// Mitsubishi GX Works2 project: MasterPlc3_2   PLC: Q03UDE

PROGRAM OUTPUT
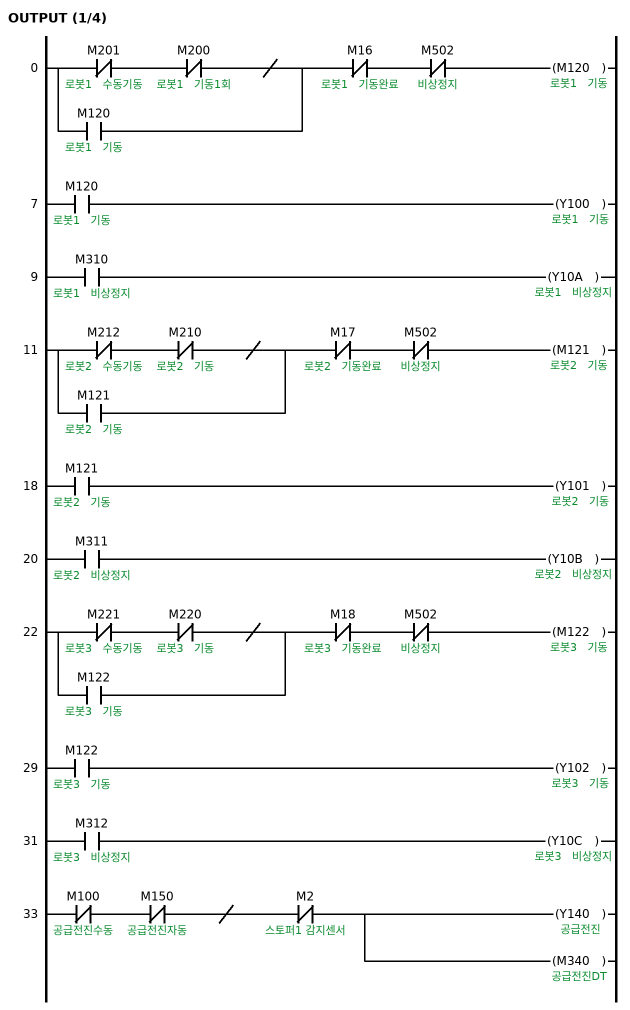
0     LDI     M201  ; 로봇1   수동기동
      ANI     M200  ; 로봇1   기동1회
      INV
      OR      M120  ; 로봇1   기동
      ANI     M16  ; 로봇1   기동완료
      ANI     M502  ; 비상정지
      OUT     M120  ; 로봇1   기동
7     LD      M120  ; 로봇1   기동
      OUT     Y100  ; 로봇1   기동
9     LD      M310  ; 로봇1   비상정지
      OUT     Y10A  ; 로봇1   비상정지
11    LDI     M212  ; 로봇2   수동기동
      ANI     M210  ; 로봇2   기동
      INV
      OR      M121  ; 로봇2   기동
      ANI     M17  ; 로봇2   기동완료
      ANI     M502  ; 비상정지
      OUT     M121  ; 로봇2   기동
18    LD      M121  ; 로봇2   기동
      OUT     Y101  ; 로봇2   기동
20    LD      M311  ; 로봇2   비상정지
      OUT     Y10B  ; 로봇2   비상정지
22    LDI     M221  ; 로봇3   수동기동
      ANI     M220  ; 로봇3   기동
      INV
      OR      M122  ; 로봇3   기동
      ANI     M18  ; 로봇3   기동완료
      ANI     M502  ; 비상정지
      OUT     M122  ; 로봇3   기동
29    LD      M122  ; 로봇3   기동
      OUT     Y102  ; 로봇3   기동
31    LD      M312  ; 로봇3   비상정지
      OUT     Y10C  ; 로봇3   비상정지
33    LDI     M100  ; 공급전진수동
      ANI     M150  ; 공급전진자동
      INV
      ANI     M2  ; 스토퍼1 감지센서
      OUT     Y140  ; 공급전진
      OUT     M340  ; 공급전진DT
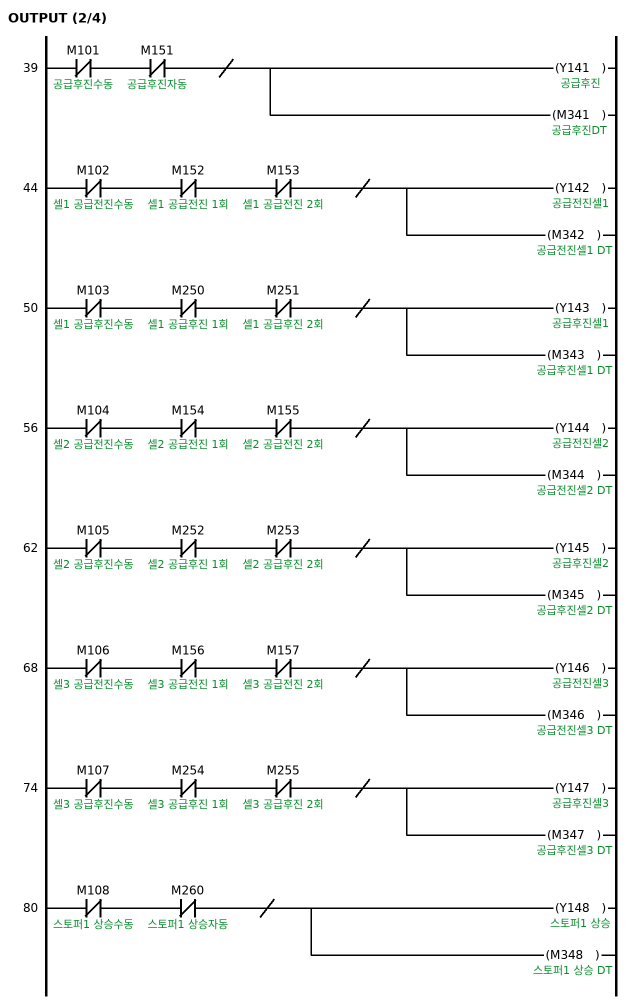
39    LDI     M101  ; 공급후진수동
      ANI     M151  ; 공급후진자동
      INV
      OUT     Y141  ; 공급후진
      OUT     M341  ; 공급후진DT
44    LDI     M102  ; 셀1 공급전진수동
      ANI     M152  ; 셀1 공급전진 1회
      ANI     M153  ; 셀1 공급전진 2회
      INV
      OUT     Y142  ; 공급전진셀1
      OUT     M342  ; 공급전진셀1 DT
50    LDI     M103  ; 셀1 공급후진수동
      ANI     M250  ; 셀1 공급후진 1회
      ANI     M251  ; 셀1 공급후진 2회
      INV
      OUT     Y143  ; 공급후진셀1
      OUT     M343  ; 공급후진셀1 DT
56    LDI     M104  ; 셀2 공급전진수동
      ANI     M154  ; 셀2 공급전진 1회
      ANI     M155  ; 셀2 공급전진 2회
      INV
      OUT     Y144  ; 공급전진셀2
      OUT     M344  ; 공급전진셀2 DT
62    LDI     M105  ; 셀2 공급후진수동
      ANI     M252  ; 셀2 공급후진 1회
      ANI     M253  ; 셀2 공급후진 2회
      INV
      OUT     Y145  ; 공급후진셀2
      OUT     M345  ; 공급후진셀2 DT
68    LDI     M106  ; 셀3 공급전진수동
      ANI     M156  ; 셀3 공급전진 1회
      ANI     M157  ; 셀3 공급전진 2회
      INV
      OUT     Y146  ; 공급전진셀3
      OUT     M346  ; 공급전진셀3 DT
74    LDI     M107  ; 셀3 공급후진수동
      ANI     M254  ; 셀3 공급후진 1회
      ANI     M255  ; 셀3 공급후진 2회
      INV
      OUT     Y147  ; 공급후진셀3
      OUT     M347  ; 공급후진셀3 DT
80    LDI     M108  ; 스토퍼1 상승수동
      ANI     M260  ; 스토퍼1 상승자동
      INV
      OUT     Y148  ; 스토퍼1 상승
      OUT     M348  ; 스토퍼1 상승 DT
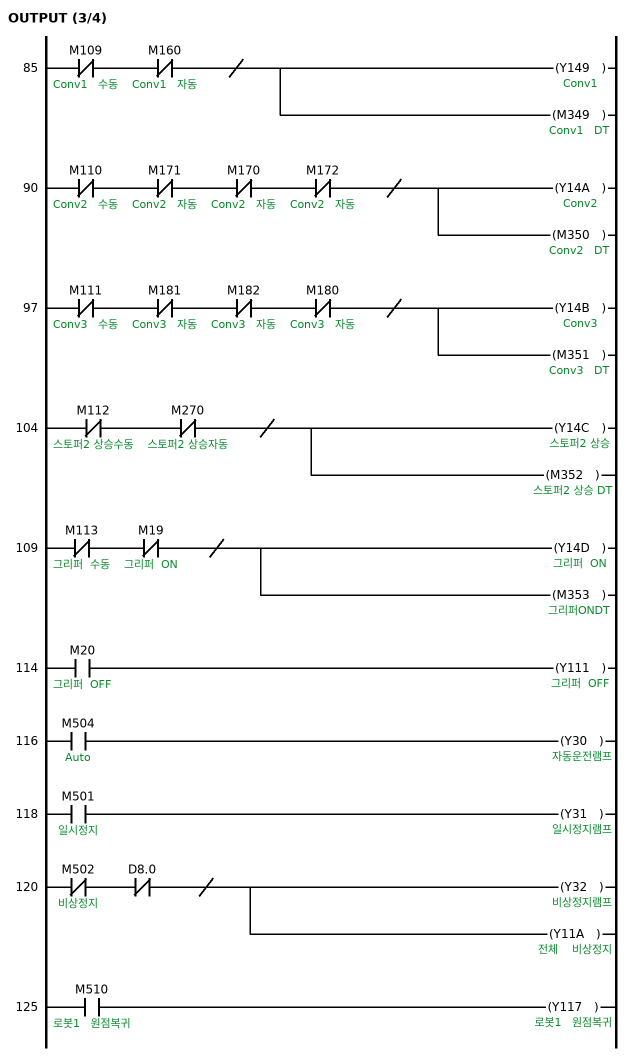
85    LDI     M109  ; Conv1   수동
      ANI     M160  ; Conv1   자동
      INV
      OUT     Y149  ; Conv1
      OUT     M349  ; Conv1   DT
90    LDI     M110  ; Conv2   수동
      ANI     M171  ; Conv2   자동
      ANI     M170  ; Conv2   자동
      ANI     M172  ; Conv2   자동
      INV
      OUT     Y14A  ; Conv2
      OUT     M350  ; Conv2   DT
97    LDI     M111  ; Conv3   수동
      ANI     M181  ; Conv3   자동
      ANI     M182  ; Conv3   자동
      ANI     M180  ; Conv3   자동
      INV
      OUT     Y14B  ; Conv3
      OUT     M351  ; Conv3   DT
104   LDI     M112  ; 스토퍼2 상승수동
      ANI     M270  ; 스토퍼2 상승자동
      INV
      OUT     Y14C  ; 스토퍼2 상승
      OUT     M352  ; 스토퍼2 상승 DT
109   LDI     M113  ; 그리퍼  수동
      ANI     M19  ; 그리퍼  ON
      INV
      OUT     Y14D  ; 그리퍼  ON
      OUT     M353  ; 그리퍼ONDT
114   LD      M20  ; 그리퍼  OFF
      OUT     Y111  ; 그리퍼  OFF
116   LD      M504  ; Auto
      OUT     Y30  ; 자동운전램프
118   LD      M501  ; 일시정지
      OUT     Y31  ; 일시정지램프
120   LDI     M502  ; 비상정지
      ANI     D8.0
      INV
      OUT     Y32  ; 비상정지램프
      OUT     Y11A  ; 전체    비상정지
125   LD      M510  ; 로봇1   원점복귀
      OUT     Y117  ; 로봇1   원점복귀
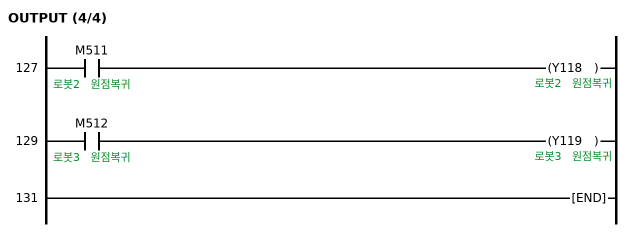
127   LD      M511  ; 로봇2   원점복귀
      OUT     Y118  ; 로봇2   원점복귀
129   LD      M512  ; 로봇3   원점복귀
      OUT     Y119  ; 로봇3   원점복귀
131   END
END_PROGRAM

PROGRAM INPUT
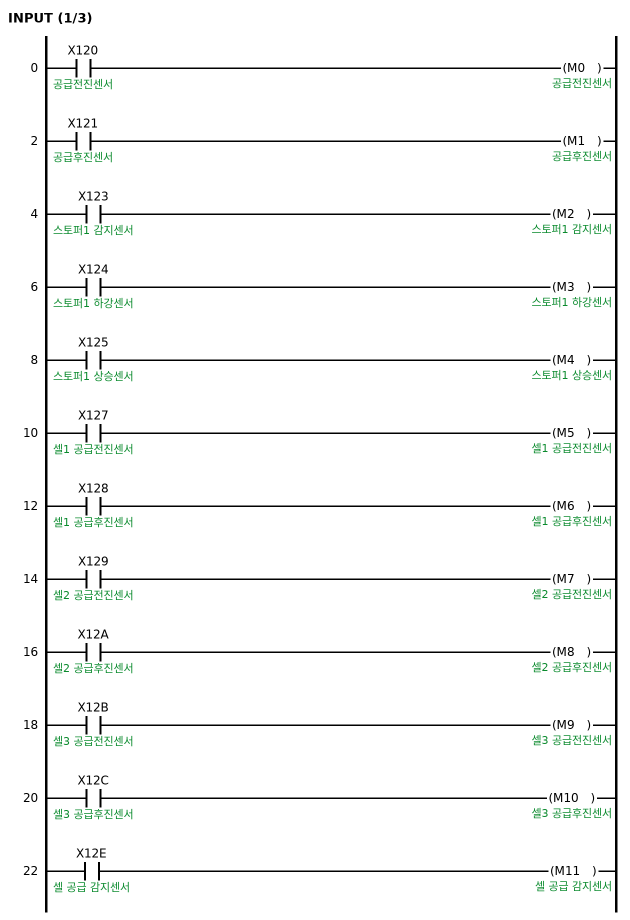
0     LD      X120  ; 공급전진센서
      OUT     M0  ; 공급전진센서
2     LD      X121  ; 공급후진센서
      OUT     M1  ; 공급후진센서
4     LD      X123  ; 스토퍼1 감지센서
      OUT     M2  ; 스토퍼1 감지센서
6     LD      X124  ; 스토퍼1 하강센서
      OUT     M3  ; 스토퍼1 하강센서
8     LD      X125  ; 스토퍼1 상승센서
      OUT     M4  ; 스토퍼1 상승센서
10    LD      X127  ; 셀1 공급전진센서
      OUT     M5  ; 셀1 공급전진센서
12    LD      X128  ; 셀1 공급후진센서
      OUT     M6  ; 셀1 공급후진센서
14    LD      X129  ; 셀2 공급전진센서
      OUT     M7  ; 셀2 공급전진센서
16    LD      X12A  ; 셀2 공급후진센서
      OUT     M8  ; 셀2 공급후진센서
18    LD      X12B  ; 셀3 공급전진센서
      OUT     M9  ; 셀3 공급전진센서
20    LD      X12C  ; 셀3 공급후진센서
      OUT     M10  ; 셀3 공급후진센서
22    LD      X12E  ; 셀 공급 감지센서
      OUT     M11  ; 셀 공급 감지센서
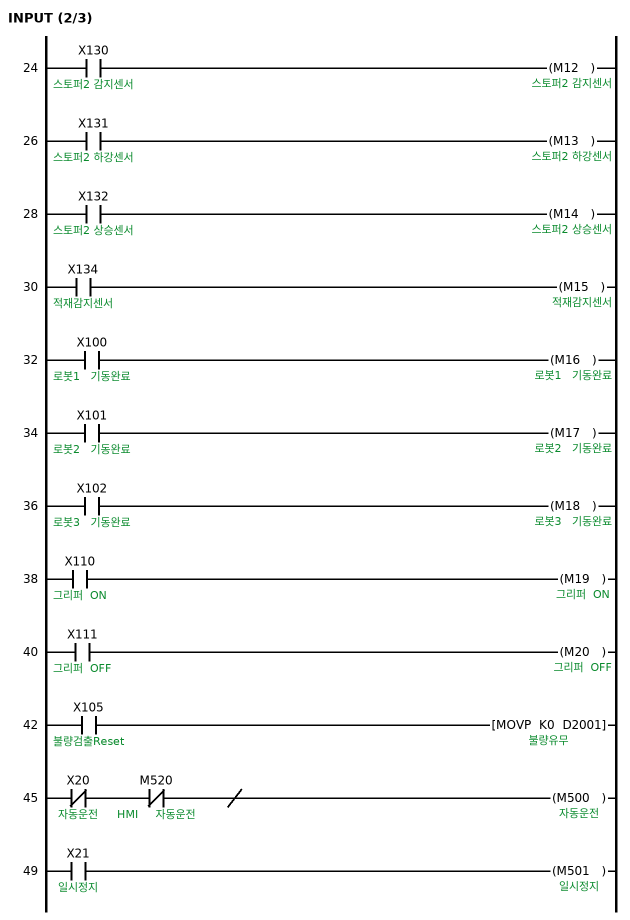
24    LD      X130  ; 스토퍼2 감지센서
      OUT     M12  ; 스토퍼2 감지센서
26    LD      X131  ; 스토퍼2 하강센서
      OUT     M13  ; 스토퍼2 하강센서
28    LD      X132  ; 스토퍼2 상승센서
      OUT     M14  ; 스토퍼2 상승센서
30    LD      X134  ; 적재감지센서
      OUT     M15  ; 적재감지센서
32    LD      X100  ; 로봇1   기동완료
      OUT     M16  ; 로봇1   기동완료
34    LD      X101  ; 로봇2   기동완료
      OUT     M17  ; 로봇2   기동완료
36    LD      X102  ; 로봇3   기동완료
      OUT     M18  ; 로봇3   기동완료
38    LD      X110  ; 그리퍼  ON
      OUT     M19  ; 그리퍼  ON
40    LD      X111  ; 그리퍼  OFF
      OUT     M20  ; 그리퍼  OFF
42    LD      X105  ; 불량검출Reset
      MOVP    K0 D2001  ; 불량유무
45    LDI     X20  ; 자동운전
      ANI     M520  ; HMI     자동운전
      INV
      OUT     M500  ; 자동운전
49    LD      X21  ; 일시정지
      OUT     M501  ; 일시정지
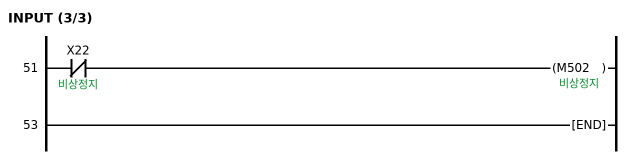
51    LDI     X22  ; 비상정지
      OUT     M502  ; 비상정지
53    END
END_PROGRAM

PROGRAM SEQUENCE
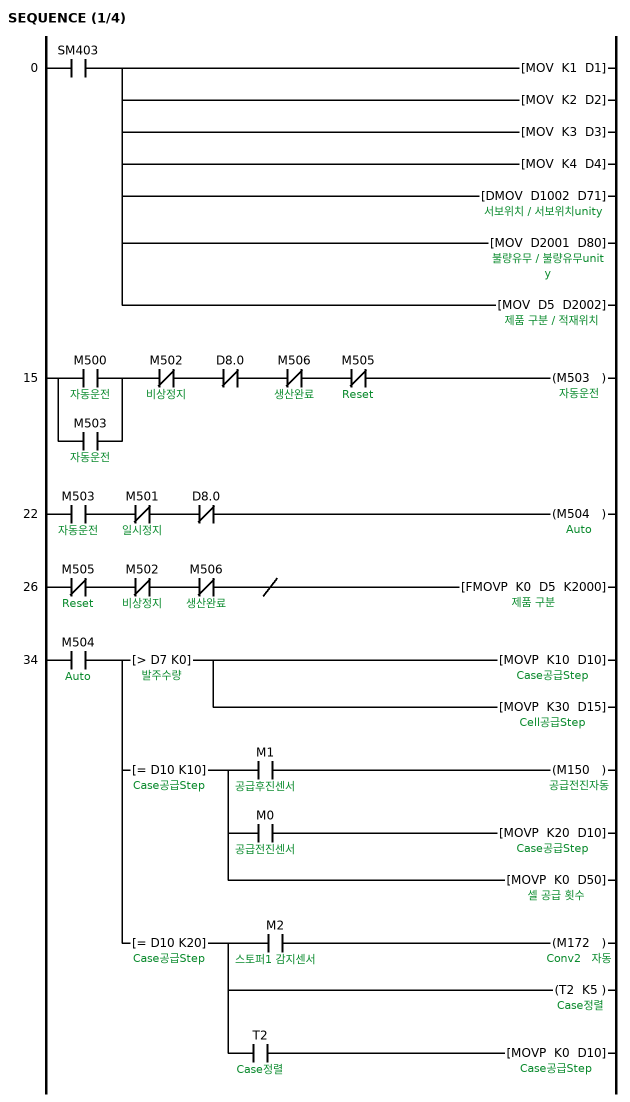
0     LD      SM403
      MOV     K1 D1
      MOV     K2 D2
      MOV     K3 D3
      MOV     K4 D4
      DMOV    D1002 D71  ; 서보위치 / 서보위치unity
      MOV     D2001 D80  ; 불량유무 / 불량유무unity
      MOV     D5 D2002  ; 제품 구분 / 적재위치
15    LD      M500  ; 자동운전
      OR      M503  ; 자동운전
      ANI     M502  ; 비상정지
      ANI     D8.0
      ANI     M506  ; 생산완료
      ANI     M505  ; Reset
      OUT     M503  ; 자동운전
22    LD      M503  ; 자동운전
      ANI     M501  ; 일시정지
      ANI     D8.0
      OUT     M504  ; Auto
26    LDI     M505  ; Reset
      ANI     M502  ; 비상정지
      ANI     M506  ; 생산완료
      INV
      FMOVP   K0 D5 K2000
34    LD      M504  ; Auto
      MPS
      AND>    D7 K0  ; 발주수량
      MOVP    K10 D10  ; Case공급Step
      MOVP    K30 D15  ; Cell공급Step
      MRD
      AND=    D10 K10  ; Case공급Step
      MPS
      AND     M1  ; 공급후진센서
      OUT     M150  ; 공급전진자동
      MRD
      AND     M0  ; 공급전진센서
      MOVP    K20 D10
      MPP
      MOVP    K0 D50  ; 셀 공급 횟수
      MPP
      AND=    D10 K20  ; Case공급Step
      MPS
      AND     M2  ; 스토퍼1 감지센서
      OUT     M172  ; Conv2   자동
      MPP
      OUT     T2 K5  ; Case정렬
      AND     T2  ; Case정렬
      MOVP    K0 D10
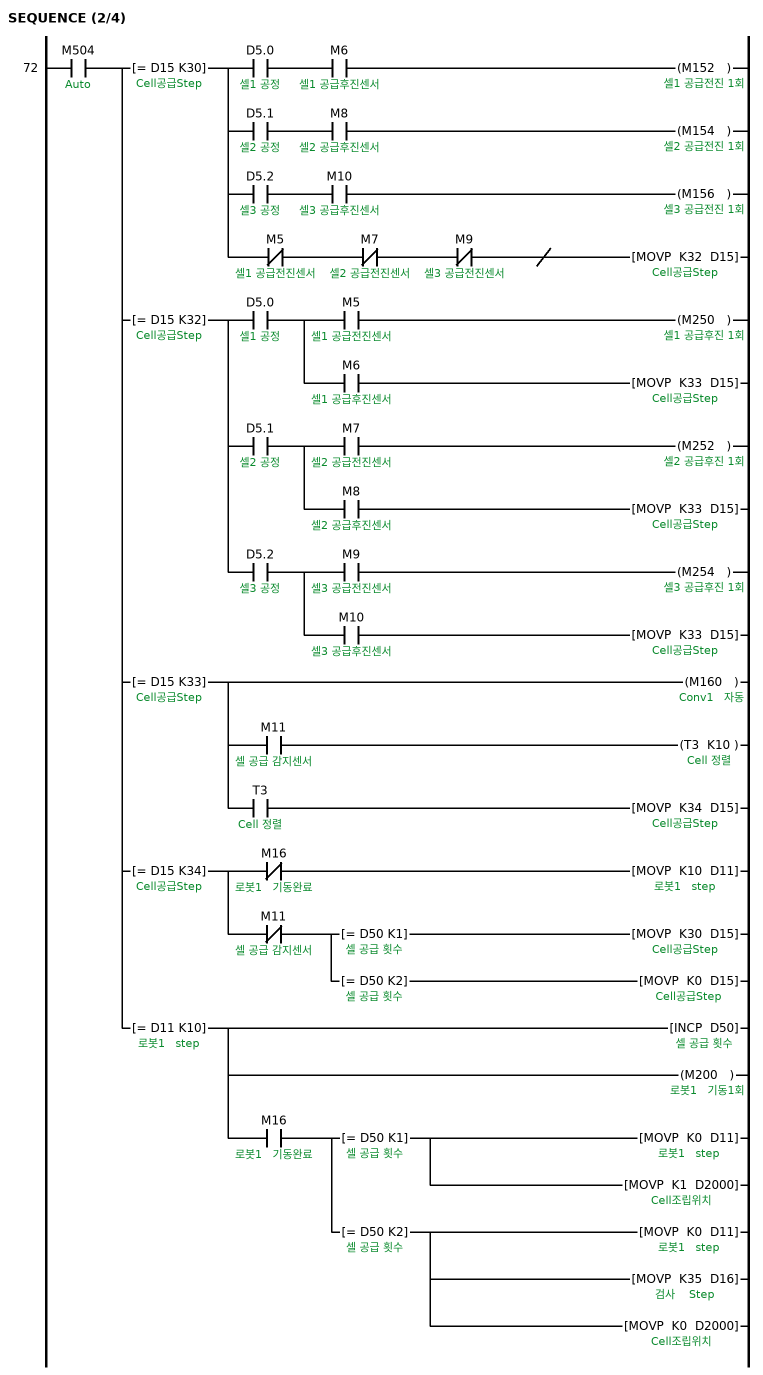
72    LD      M504  ; Auto
      MPS
      AND=    D15 K30  ; Cell공급Step
      MPS
      AND     D5.0  ; 셀1 공정
      AND     M6  ; 셀1 공급후진센서
      OUT     M152  ; 셀1 공급전진 1회
      MRD
      AND     D5.1  ; 셀2 공정
      AND     M8  ; 셀2 공급후진센서
      OUT     M154  ; 셀2 공급전진 1회
      MRD
      AND     D5.2  ; 셀3 공정
      AND     M10  ; 셀3 공급후진센서
      OUT     M156  ; 셀3 공급전진 1회
      MPP
      ANI     M5  ; 셀1 공급전진센서
      ANI     M7  ; 셀2 공급전진센서
      ANI     M9  ; 셀3 공급전진센서
      INV
      MOVP    K32 D15
      MRD
      AND=    D15 K32  ; Cell공급Step
      MPS
      AND     D5.0  ; 셀1 공정
      MPS
      AND     M5  ; 셀1 공급전진센서
      OUT     M250  ; 셀1 공급후진 1회
      MPP
      AND     M6  ; 셀1 공급후진센서
      MOVP    K33 D15
      MRD
      AND     D5.1  ; 셀2 공정
      MPS
      AND     M7  ; 셀2 공급전진센서
      OUT     M252  ; 셀2 공급후진 1회
      MPP
      AND     M8  ; 셀2 공급후진센서
      MOVP    K33 D15
      MPP
      AND     D5.2  ; 셀3 공정
      MPS
      AND     M9  ; 셀3 공급전진센서
      OUT     M254  ; 셀3 공급후진 1회
      MPP
      AND     M10  ; 셀3 공급후진센서
      MOVP    K33 D15
      MRD
      AND=    D15 K33  ; Cell공급Step
      OUT     M160  ; Conv1   자동
      MPS
      AND     M11  ; 셀 공급 감지센서
      OUT     T3 K10  ; Cell 정렬
      MPP
      AND     T3  ; Cell 정렬
      MOVP    K34 D15
      MRD
      AND=    D15 K34  ; Cell공급Step
      MPS
      ANI     M16  ; 로봇1   기동완료
      MOVP    K10 D11  ; 로봇1   step
      MPP
      ANI     M11  ; 셀 공급 감지센서
      MPS
      AND=    D50 K1  ; 셀 공급 횟수
      MOVP    K30 D15
      MPP
      AND=    D50 K2  ; 셀 공급 횟수
      MOVP    K0 D15
      MPP
      AND=    D11 K10  ; 로봇1   step
      INCP    D50
      OUT     M200  ; 로봇1   기동1회
      AND     M16  ; 로봇1   기동완료
      MPS
      AND=    D50 K1  ; 셀 공급 횟수
      MOVP    K0 D11
      MOVP    K1 D2000  ; Cell조립위치
      MPP
      AND=    D50 K2  ; 셀 공급 횟수
      MOVP    K0 D11
      MOVP    K35 D16  ; 검사    Step
      MOVP    K0 D2000
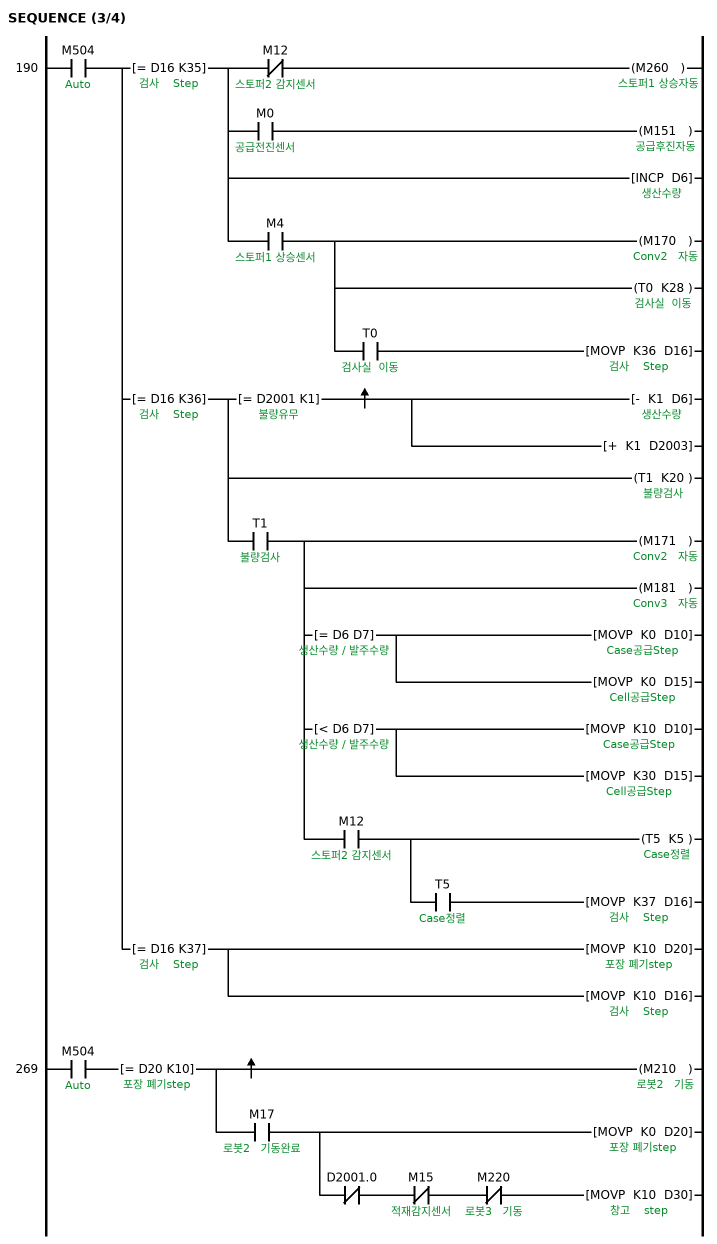
190   LD      M504  ; Auto
      MPS
      AND=    D16 K35  ; 검사    Step
      MPS
      ANI     M12  ; 스토퍼2 감지센서
      OUT     M260  ; 스토퍼1 상승자동
      MRD
      AND     M0  ; 공급전진센서
      OUT     M151  ; 공급후진자동
      MPP
      INCP    D6  ; 생산수량
      AND     M4  ; 스토퍼1 상승센서
      OUT     M170  ; Conv2   자동
      OUT     T0 K28  ; 검사실  이동
      AND     T0  ; 검사실  이동
      MOVP    K36 D16
      MRD
      AND=    D16 K36  ; 검사    Step
      MPS
      AND=    D2001 K1  ; 불량유무
      MEP
      -       K1 D6
      +       K1 D2003
      MPP
      OUT     T1 K20  ; 불량검사
      AND     T1  ; 불량검사
      OUT     M171  ; Conv2   자동
      OUT     M181  ; Conv3   자동
      MPS
      AND=    D6 D7  ; 생산수량 / 발주수량
      MOVP    K0 D10
      MOVP    K0 D15
      MRD
      AND<    D6 D7  ; 생산수량 / 발주수량
      MOVP    K10 D10
      MOVP    K30 D15
      MPP
      AND     M12  ; 스토퍼2 감지센서
      OUT     T5 K5  ; Case정렬
      AND     T5  ; Case정렬
      MOVP    K37 D16
      MPP
      AND=    D16 K37  ; 검사    Step
      MOVP    K10 D20  ; 포장 폐기step
      MOVP    K10 D16
269   LD      M504  ; Auto
      AND=    D20 K10  ; 포장 폐기step
      MPS
      MEP
      OUT     M210  ; 로봇2   기동
      MPP
      AND     M17  ; 로봇2   기동완료
      MOVP    K0 D20
      ANI     D2001.0
      ANI     M15  ; 적재감지센서
      ANI     M220  ; 로봇3   기동
      MOVP    K10 D30  ; 창고    step
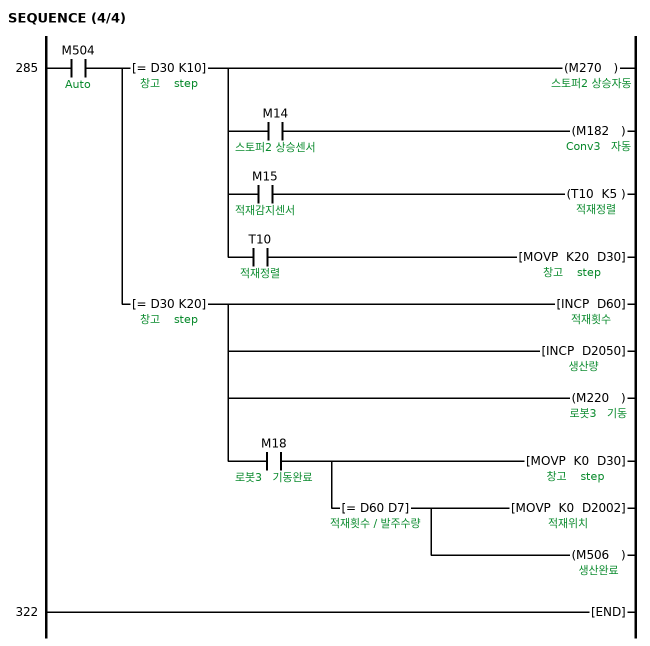
285   LD      M504  ; Auto
      MPS
      AND=    D30 K10  ; 창고    step
      OUT     M270  ; 스토퍼2 상승자동
      MPS
      AND     M14  ; 스토퍼2 상승센서
      OUT     M182  ; Conv3   자동
      MRD
      AND     M15  ; 적재감지센서
      OUT     T10 K5  ; 적재정렬
      MPP
      AND     T10  ; 적재정렬
      MOVP    K20 D30
      MPP
      AND=    D30 K20  ; 창고    step
      INCP    D60  ; 적재횟수
      INCP    D2050  ; 생산량
      OUT     M220  ; 로봇3   기동
      AND     M18  ; 로봇3   기동완료
      MOVP    K0 D30
      AND=    D60 D7  ; 적재횟수 / 발주수량
      MOVP    K0 D2002
      OUT     M506  ; 생산완료
322   END
END_PROGRAM

// device comments not shown above
M521  ; HMI     일시정지
M522  ; HMI     비상정지
Y21A  ; 로봇    비상정지
D8  ; 비상정지
D2051  ; 불량수량
D6.0  ; 양품
D6.1  ; 불량
D8.1  ; 조립    Step
D8.2  ; 로봇1   step
